FUNCTION_BLOCK CM_Actuator2State
VAR_INPUT
	CM_Number : INT;
	
	IN_MANUAL :BOOL;
	IN_AUTO : BOOL;
	
	IN_HMI_HAND : BOOL;
	
	IN_MANUAL_ON : BOOL;
	IN_AUTO_ON : BOOL;
	
	IN_OFF : BOOL;
	
	IN_AlarmHigh_Enable : BOOL;
	IN_AlarmLow_Enable : BOOL;
	IN_AlarmDelay_H : INT;
	IN_AlarmDelay_L : INT;
	
	IN_Alarm_Condition_H : BOOL;
	IN_Alarm_Condition_L : BOOL;
	
	IN_CM_Interlock : BOOL;
	
END_VAR
VAR_OUTPUT
	
	AUTO_ON :BOOL;
	HMI_HAND_ON : BOOL;
	
	OUT_ON : BOOL;
	OUT_OFF :BOOL;
	
	
	PO_ALARM_H : BOOL;
	PO_ALARM_L : BOOL;;
	
	PO_Interlocked : BOOL;
	
END_VAR
VAR
	SR_Auto: SR;
	
	prg_scan_H : INT; // used for alarm delay
	prg_scan_L : INT; // used for alarm delay
	
	Alarm_limit_Exceeded_H : BOOL;
	Alarm_limit_Exceeded_L : BOOL;
	
	Alarm_Ack_H : BOOL;
	Alarm_Ack_L : BOOL;
END_VAR
VAR_IN_OUT
	CM_UDT_CTRL : Udt_CM_Actuator2State;
	Plant_control : Udt_PlantControl;
END_VAR
VAR // added by the converter: edge detectors and wires of the graphical bodies
    _w1, _w2 : BOOL;
END_VAR

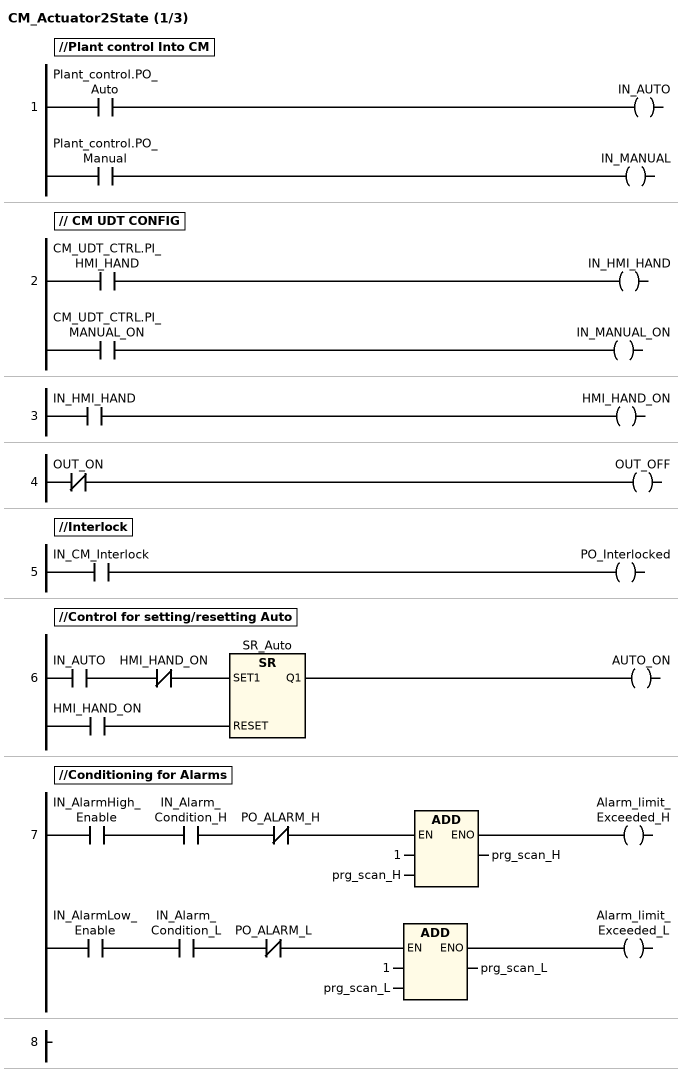
// NETWORK 1
// label: //Plant control Into CM
IN_AUTO := Plant_control.PO_Auto;
IN_MANUAL := Plant_control.PO_Manual;

// NETWORK 2
// label: // CM UDT CONFIG
IN_HMI_HAND := CM_UDT_CTRL.PI_HMI_HAND;
IN_MANUAL_ON := CM_UDT_CTRL.PI_MANUAL_ON;

// NETWORK 3
HMI_HAND_ON := IN_HMI_HAND;

// NETWORK 4
OUT_OFF := NOT OUT_ON;

// NETWORK 5
// label: //Interlock
PO_Interlocked := IN_CM_Interlock;

// NETWORK 6
// label: //Control for setting/resetting Auto
SR_Auto(SET1 := IN_AUTO AND NOT HMI_HAND_ON, RESET := HMI_HAND_ON); // SR
AUTO_ON := SR_Auto.Q1;

// NETWORK 7
// label: //Conditioning for Alarms
_w1 := IN_AlarmHigh_Enable AND IN_Alarm_Condition_H AND NOT PO_ALARM_H;
IF _w1 THEN prg_scan_H := 1 + prg_scan_H; END_IF
Alarm_limit_Exceeded_H := _w1;
_w2 := IN_AlarmLow_Enable AND IN_Alarm_Condition_L AND NOT PO_ALARM_L;
IF _w2 THEN prg_scan_L := 1 + prg_scan_L; END_IF
Alarm_limit_Exceeded_L := _w2;

// NETWORK 8

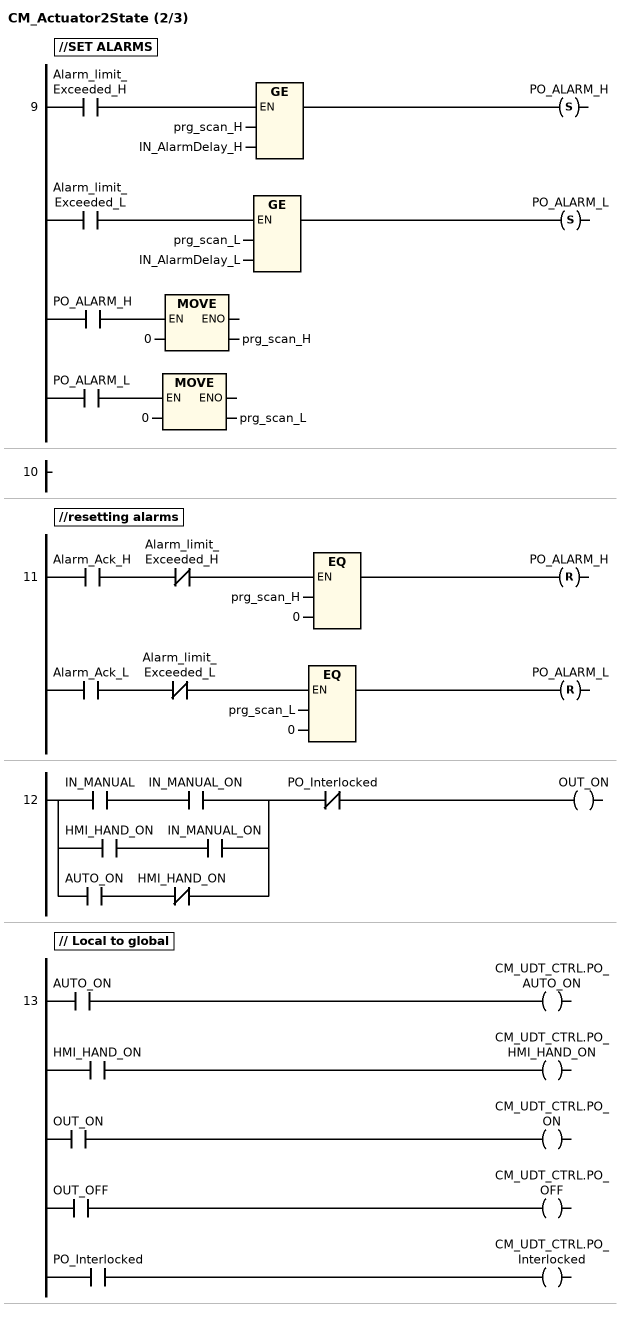
// NETWORK 9
// label: //SET ALARMS
PO_ALARM_H S= Alarm_limit_Exceeded_H AND prg_scan_H >= IN_AlarmDelay_H;
PO_ALARM_L S= Alarm_limit_Exceeded_L AND prg_scan_L >= IN_AlarmDelay_L;
IF PO_ALARM_H THEN prg_scan_H := 0; END_IF
IF PO_ALARM_L THEN prg_scan_L := 0; END_IF

// NETWORK 10

// NETWORK 11
// label: //resetting alarms
PO_ALARM_H R= Alarm_Ack_H AND NOT Alarm_limit_Exceeded_H AND prg_scan_H = 0;
PO_ALARM_L R= Alarm_Ack_L AND NOT Alarm_limit_Exceeded_L AND prg_scan_L = 0;

// NETWORK 12
OUT_ON := (IN_MANUAL AND IN_MANUAL_ON OR HMI_HAND_ON AND IN_MANUAL_ON OR AUTO_ON AND NOT HMI_HAND_ON) AND NOT PO_Interlocked;

// NETWORK 13
// label: // Local to global
CM_UDT_CTRL.PO_AUTO_ON := AUTO_ON;
CM_UDT_CTRL.PO_HMI_HAND_ON := HMI_HAND_ON;
CM_UDT_CTRL.PO_ON := OUT_ON;
CM_UDT_CTRL.PO_OFF := OUT_OFF;
CM_UDT_CTRL.PO_Interlocked := PO_Interlocked;

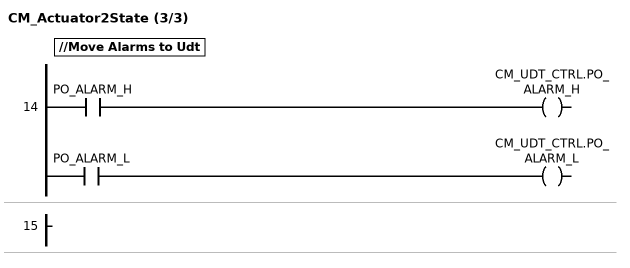
// NETWORK 14
// label: //Move Alarms to Udt
CM_UDT_CTRL.PO_ALARM_H := PO_ALARM_H;
CM_UDT_CTRL.PO_ALARM_L := PO_ALARM_L;

// NETWORK 15

END_FUNCTION_BLOCK

(* stored: Version 1.1.0.1, ProductVersion 3.1.4024.13
   POU CM_Actuator2State: Id {748b01c6-4635-4913-9fe9-6b85d8a796d7}, SpecialFunc None *)
